TYPE "WkClockSet"
VERSION : 0.1
// Block: WkClockSet
   STRUCT
      Set_ON : Time_Of_Day;
      Set_OFF : Time_Of_Day;
      Enable : Bool;
   END_STRUCT;

END_TYPE
